(* IEC 61131-3 sources: AXOpen/src/components.dukane.welders/app/SystemConstants, 2 files *)

(* ---- plc_line_IoAddresses.st ---- *)
CONFIGURATION IoAddresses
    VAR_GLOBAL

        // Module dukaneiqauto/iQ_to_PLC_Inputs
        dukaneiqauto_iQ_to_PLC_Inputs_Input AT %IB0 : dukaneiqauto_iQ_to_PLC_Inputs_Input_Layout;

        // Module dukaneiqauto/PLC_to_iQ_Outputs
        dukaneiqauto_PLC_to_iQ_Outputs_Output AT %QB0 : dukaneiqauto_PLC_to_iQ_Outputs_Output_Layout;
    END_VAR
END_CONFIGURATION

TYPE
    dukaneiqauto_iQ_to_PLC_Inputs_Input_Layout : STRUCT
        Signals_0 AT %B0 : DWORD;
        Signals_1 AT %B4 : DWORD;
        Signals_2 AT %B8 : DWORD;
        Signals_3 AT %B12 : DWORD;
        Signals_4 AT %B16 : DWORD;
        Signals_5 AT %B20 : DWORD;
        Signals_6 AT %B24 : DWORD;
        Signals_7 AT %B28 : DWORD;
        Signals_8 AT %B32 : DWORD;
        Signals_9 AT %B36 : DWORD;
        Signals_10 AT %B40 : DWORD;
        Signals_11 AT %B44 : DWORD;
        Signals_12 AT %B48 : DWORD;
        Signals_13 AT %B52 : DWORD;
        Signals_14 AT %B56 : DWORD;
        Signals_15 AT %B60 : DWORD;
        Signals_16 AT %B64 : DWORD;
        Signals_17 AT %B68 : DWORD;
        Signals_18 AT %B72 : DWORD;
        Signals_19 AT %B76 : DWORD;
        Signals_20 AT %B80 : DWORD;
        Signals_21 AT %B84 : DWORD;
        Signals_22 AT %B88 : DWORD;
        Signals_23 AT %B92 : DWORD;
        Signals_24 AT %B96 : DWORD;
        Signals_25 AT %B100 : DWORD;
        Signals_26 AT %B104 : DWORD;
        Signals_27 AT %B108 : DWORD;
        Signals_28 AT %B112 : DWORD;
        Signals_29 AT %B116 : DWORD;
        Signals_30 AT %B120 : DWORD;
        Signals_31 AT %B124 : DWORD;
        Signals_32 AT %B128 : DWORD;
        Signals_33 AT %B132 : DWORD;
        Signals_34 AT %B136 : DWORD;
    END_STRUCT;
END_TYPE

TYPE
    dukaneiqauto_PLC_to_iQ_Outputs_Output_Layout : STRUCT
        Signals_0 AT %B0 : DWORD;
        Signals_1 AT %B4 : DWORD;
        Signals_2 AT %B8 : DWORD;
        Signals_3 AT %B12 : DWORD;
        Signals_4 AT %B16 : DWORD;
    END_STRUCT;
END_TYPE

(* ---- plc_line_HwIdentifiers.st ---- *)
CONFIGURATION HardwareIDs
    VAR_GLOBAL CONSTANT
        dukaneiqauto_HwID : UINT := UINT#258;
        dukaneiqauto_PLC_to_iQ_Outputs_PLC_to_iQ_Outputs_HwID : UINT := UINT#263;
        dukaneiqauto_Rack_HwID : UINT := UINT#261;
        dukaneiqauto_dukaneiqauto_HwID : UINT := UINT#262;
        dukaneiqauto_dukaneiqauto_DAP_HwID : UINT := UINT#265;
        dukaneiqauto_dukaneiqauto_Interface_HwID : UINT := UINT#257;
        dukaneiqauto_dukaneiqauto_Interface_Port_1_HwID : UINT := UINT#259;
        dukaneiqauto_dukaneiqauto_Interface_Port_2_HwID : UINT := UINT#260;
        dukaneiqauto_iQ_to_PLC_Inputs_iQ_to_PLC_Inputs_HwID : UINT := UINT#264;
        plc_line_HwID : UINT := UINT#32;
        plc_line_Rail_0_HwID : UINT := UINT#266;
        plc_line_plc_line_HwID : UINT := UINT#48;
        plc_line_plc_line_CPU_display_1_HwID : UINT := UINT#54;
        plc_line_plc_line_Card_reader_writer_1_HwID : UINT := UINT#51;
        plc_line_plc_line_DP_interface_1_HwID : UINT := UINT#60;
        plc_line_plc_line_OPC_UA_1_HwID : UINT := UINT#117;
        plc_line_plc_line_PROFINET_interface_1_HwID : UINT := UINT#64;
        plc_line_plc_line_PROFINET_interface_1_Port_1_HwID : UINT := UINT#65;
        plc_line_plc_line_PROFINET_interface_1_Port_2_HwID : UINT := UINT#66;
        plc_line_plc_line_PROFINET_interface_2_HwID : UINT := UINT#72;
        plc_line_plc_line_PROFINET_interface_2_Port_3_HwID : UINT := UINT#73;
        plc_line_plc_line_Virtual_communication_interface_HwID : UINT := UINT#135;
        profinet_plc_line_HwID : UINT := UINT#256;

    END_VAR
END_CONFIGURATION
